{library PUBLIC}

(* Sequence for a specific communicator during send or receive *)
TYPE DATAGRAM_SEQUENCE : (
	DATAGRAM_SEQUENCE_ERROR:=-1,
	DATAGRAM_SEQUENCE_INIT:=-0,
	DATAGRAM_SEQUENCE_NOP,							(* No operation - free *)
	DATAGRAM_SEQUENCE_INIT_SEND,
	DATAGRAM_SEQUENCE_SEND_1,
	DATAGRAM_SEQUENCE_SEND_2,
	DATAGRAM_SEQUENCE_SEND_3,

	DATAGRAM_SEQUENCE_INIT_RECEIVE,
	DATAGRAM_SEQUENCE_RECEIVE_1,
	DATAGRAM_SEQUENCE_RECEIVE_2,
	DATAGRAM_SEQUENCE_RECEIVE_3,

	DATAGRAM_SEQUENCE_DONE
);
END_TYPE
//  DATAGRAM_SEQUENCE_ERROR = '-1'
//  DATAGRAM_SEQUENCE_INIT = '-0'

(* stored: Version 1.1.0.1, ProductVersion 3.1.4024.2
   EnumerationTextList DATAGRAM_SEQUENCE: Id {6270b8ff-9595-4672-8fc7-e5feb0d2e155} *)
